% RSLogix 500 project P6_ABIOLA_A V3_BAK025.RSS, saved by version 8.30.00.16 %
PROJECT "UNTITLED"    % processor: Bul.1763 MicroLogix 1100 Series B %

PROGRAM FILES
  LAD 2 "PROG LOGIC"  6 rungs
  LAD 3 "I/O"  2 rungs  % Contains all the input and output devices used %

DATA FILES
  O0 OUTPUT  4 elements
  I1 INPUT  6 elements
  S2 STATUS  66 elements
  B3 BINARY  1 elements
  T4 TIMER  1 elements
  C5 COUNTER  1 elements
  R6 CONTROL  1 elements
  N7 INTEGER  4 elements
  F8 FLOAT  1 elements

LADDER 2 "PROG LOGIC"
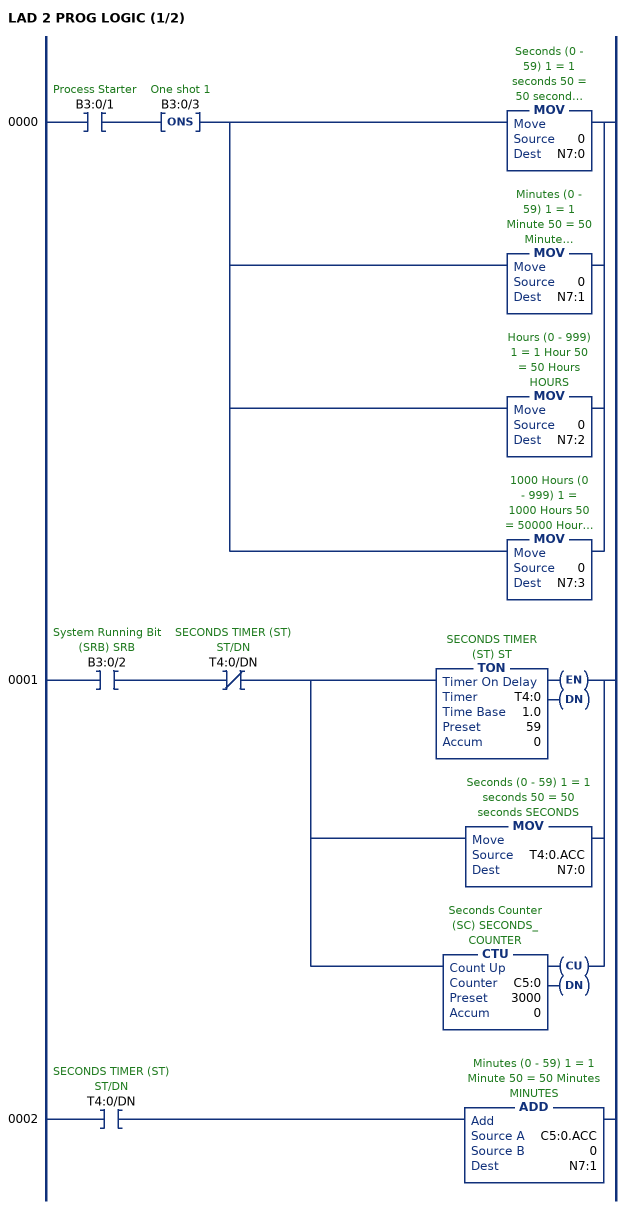
% Rung: 0 %
SOR XIC B3:0/1 ONS B3:0/3 BST MOV 0 N7:0 NXB BST MOV 0 N7:1 NXB BST MOV 0 N7:2 NXB MOV 0 N7:3 BND BND BND EOR
%   B3:0/1  "Process Starter" %
%   B3:0/3  "One shot 1" %
%   N7:0  SECONDS  "Seconds (0 - 59) 1 = 1 seconds 50 = 50 seconds" %
%   N7:1  MINUTES  "Minutes (0 - 59) 1 = 1 Minute 50 = 50 Minutes" %
%   N7:2  HOURS  "Hours (0 - 999) 1 = 1 Hour 50 = 50 Hours" %
%   N7:3  HOURS_1000  "1000 Hours (0 - 999) 1 = 1000 Hours 50 = 50000 Hours" %
% Rung: 1 %
SOR XIC B3:0/2 XIO T4:0/DN BST BST TON T4:0 1.0 59 0 NXB MOV T4:0.ACC N7:0 BND NXB CTU C5:0 3000 0 BND EOR
%   B3:0/2  SRB  "System Running Bit (SRB)" %
%   T4:0  ST  "SECONDS TIMER (ST)" %
%   N7:0  SECONDS  "Seconds (0 - 59) 1 = 1 seconds 50 = 50 seconds" %
%   C5:0  SECONDS_COUNTER  "Seconds Counter (SC)" %
% Rung: 2 %
SOR XIC T4:0/DN ADD C5:0.ACC 0 N7:1 EOR
%   T4:0  ST  "SECONDS TIMER (ST)" %
%   C5:0  SECONDS_COUNTER  "Seconds Counter (SC)" %
%   N7:1  MINUTES  "Minutes (0 - 59) 1 = 1 Minute 50 = 50 Minutes" %

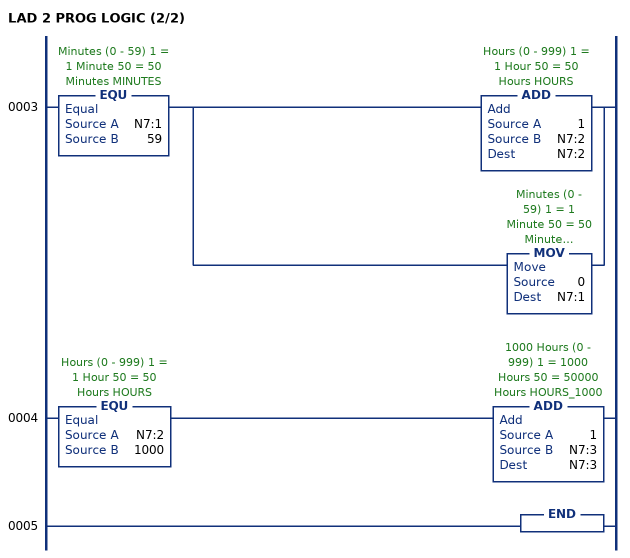
% Rung: 3 %
SOR EQU N7:1 59 BST ADD 1 N7:2 N7:2 NXB MOV 0 N7:1 BND EOR
%   N7:1  MINUTES  "Minutes (0 - 59) 1 = 1 Minute 50 = 50 Minutes" %
%   N7:2  HOURS  "Hours (0 - 999) 1 = 1 Hour 50 = 50 Hours" %
% Rung: 4 %
SOR EQU N7:2 1000 ADD 1 N7:3 N7:3 EOR
%   N7:2  HOURS  "Hours (0 - 999) 1 = 1 Hour 50 = 50 Hours" %
%   N7:3  HOURS_1000  "1000 Hours (0 - 999) 1 = 1000 Hours 50 = 50000 Hours" %
% Rung: 5 %
SOR END EOR

LADDER 3 "I/O"    % Contains all the input and output devices used %
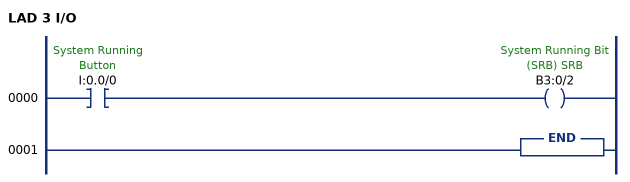
% Rung: 0 %
SOR XIC I:0.0/0 OTE B3:0/2 EOR
%   I:0.0/0  "System Running Button" %
%   B3:0/2  SRB  "System Running Bit (SRB)" %
% Rung: 1 %
SOR END EOR

DATA TABLE (non-zero values as saved)
DATA T4
% .PRE .ACC %
% T4:0 % 59 0
DATA C5
% .PRE .ACC %
% C5:0 % 3000 0
